# EPICS substitutions: evrSupport/Db/ioc/IOC-LI21-IM01trig.substitutions
# Trigger records - Current Monitor (IM) EVR:IN20:IM01, IOC:IN20:IM01; Devices are in LI21
#
# refer to Sharepoint document: Controls | Timing | timingTriggers.xls
#
# Must also have pattern records
# Note: WID, DES, TEC are in terms of nSec and are unique per device
#
file evrDevTrig.db {
#      Device	      , Description   , EVR  ,  width ,desired  , EC delay  , EVR  , EVR,  IOC          , slope
#			                            Trigger       wrt TREF   wrt fiducial loca   unit                 1/119Mhz
  pattern { DEV       ,  DESC         , T    ,  WID   , DES     , TEC       , LOCA , UNIT, IOC          , ESLO
                      ,  PREC         , EGU  ,  DRVL  , DRVH    , EVG       , OTP}
	  { TORO:LI21:205:,  "IMBC1l"     , 3    ,  100   , 10      , LCLSHOME  , IN20 , IM01, IOC:IN20:IM01, 8.40336692324359
                      ,  1            ,"nSec", -2.8E06, 2.8E06  , IN20:EV01 , OTP3}
	  { TORO:LI21:277:,  "IMBC1O"     , 4    ,  100   , 10      , LCLSHOME  , IN20 , IM01, IOC:IN20:IM01, 8.40336692324359
                      ,  1            ,"nSec", -2.8E06, 2.8E06  , IN20:EV01 , OTP4}

}
